// Mitsubishi GX Works2 project: TSUNE-14.10.2020_Q03UDV-FR   PLC: Q03UDV

PROGRAM MAIN
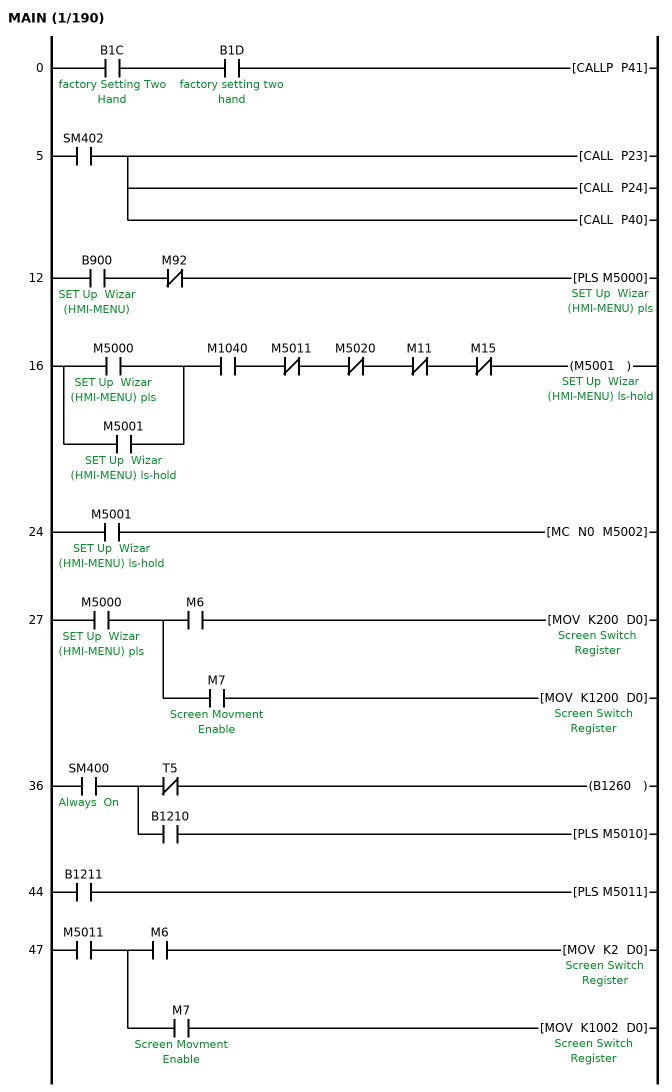
0     LD      B1C  ; factory Setting Two Hand
      AND     B1D  ; factory setting two hand
      CALLP   P41
5     LD      SM402
      CALL    P23
      CALL    P24
      CALL    P40
12    LD      B900  ; SET Up  Wizar  (HMI-MENU)
      ANI     M92
      PLS     M5000  ; SET Up  Wizar  (HMI-MENU) pls
16    LD      M5000  ; SET Up  Wizar  (HMI-MENU) pls
      OR      M5001  ; SET Up  Wizar (HMI-MENU) ls-hold
      AND     M1040
      ANI     M5011
      ANI     M5020
      ANI     M11
      ANI     M15
      OUT     M5001  ; SET Up  Wizar (HMI-MENU) ls-hold
24    LD      M5001  ; SET Up  Wizar (HMI-MENU) ls-hold
      MC      N0 M5002
27    LD      M5000  ; SET Up  Wizar  (HMI-MENU) pls
      MPS
      AND     M6
      MOV     K200 D0  ; Screen Switch Register
      MPP
      AND     M7  ; Screen Movment Enable
      MOV     K1200 D0
36    LD      SM400  ; Always  On
      MPS
      ANI     T5
      OUT     B1260
      MPP
      AND     B1210
      PLS     M5010
44    LD      B1211
      PLS     M5011
47    LD      M5011
      MPS
      AND     M6
      MOV     K2 D0
      MPP
      AND     M7  ; Screen Movment Enable
      MOV     K1002 D0
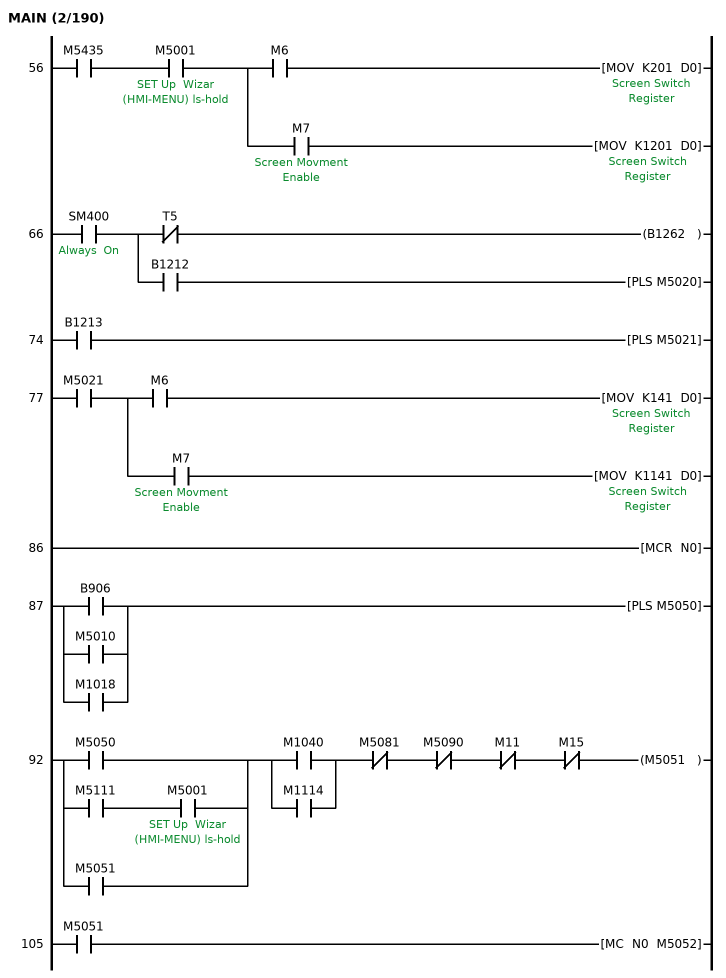
56    LD      M5435
      AND     M5001  ; SET Up  Wizar (HMI-MENU) ls-hold
      MPS
      AND     M6
      MOV     K201 D0
      MPP
      AND     M7  ; Screen Movment Enable
      MOV     K1201 D0
66    LD      SM400  ; Always  On
      MPS
      ANI     T5
      OUT     B1262
      MPP
      AND     B1212
      PLS     M5020
74    LD      B1213
      PLS     M5021
77    LD      M5021
      MPS
      AND     M6
      MOV     K141 D0
      MPP
      AND     M7  ; Screen Movment Enable
      MOV     K1141 D0
86    MCR     N0
87    LD      B906
      OR      M5010
      OR      M1018
      PLS     M5050
92    LD      M5050
      LD      M5111
      AND     M5001  ; SET Up  Wizar (HMI-MENU) ls-hold
      ORB
      OR      M5051
      LD      M1040
      OR      M1114
      ANB
      ANI     M5081
      ANI     M5090
      ANI     M11
      ANI     M15
      OUT     M5051
105   LD      M5051
      MC      N0 M5052
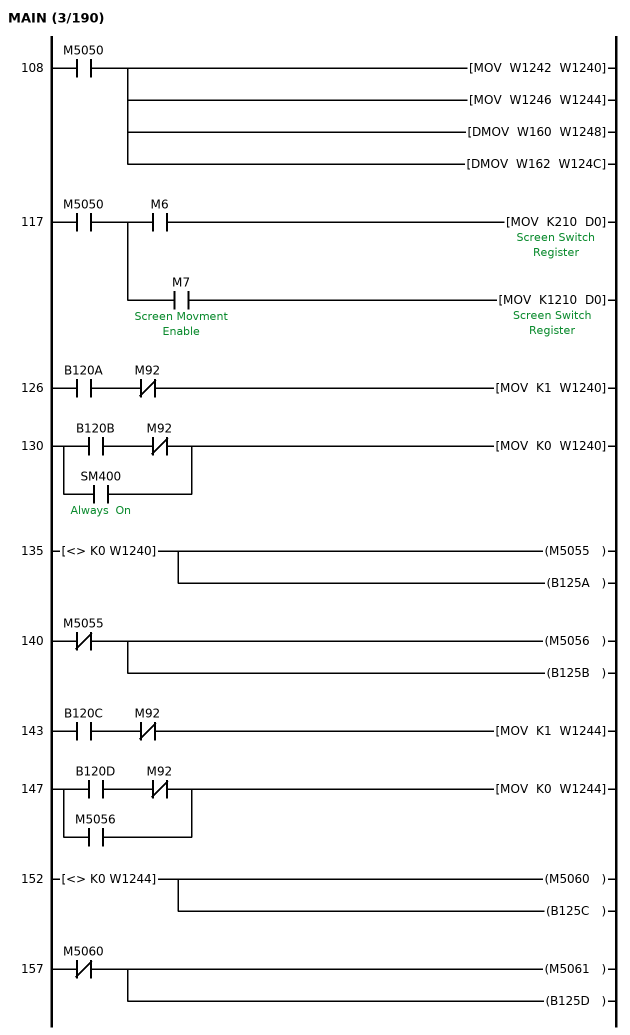
108   LD      M5050
      MOV     W1242 W1240
      MOV     W1246 W1244
      DMOV    W160 W1248
      DMOV    W162 W124C
117   LD      M5050
      MPS
      AND     M6
      MOV     K210 D0
      MPP
      AND     M7  ; Screen Movment Enable
      MOV     K1210 D0
126   LD      B120A
      ANI     M92
      MOV     K1 W1240
130   LD      B120B
      ANI     M92
      OR      SM400  ; Always  On
      MOV     K0 W1240
135   LD<>    K0 W1240
      OUT     M5055
      OUT     B125A
140   LDI     M5055
      OUT     M5056
      OUT     B125B
143   LD      B120C
      ANI     M92
      MOV     K1 W1244
147   LD      B120D
      ANI     M92
      OR      M5056
      MOV     K0 W1244
152   LD<>    K0 W1244
      OUT     M5060
      OUT     B125C
157   LDI     M5060
      OUT     M5061
      OUT     B125D
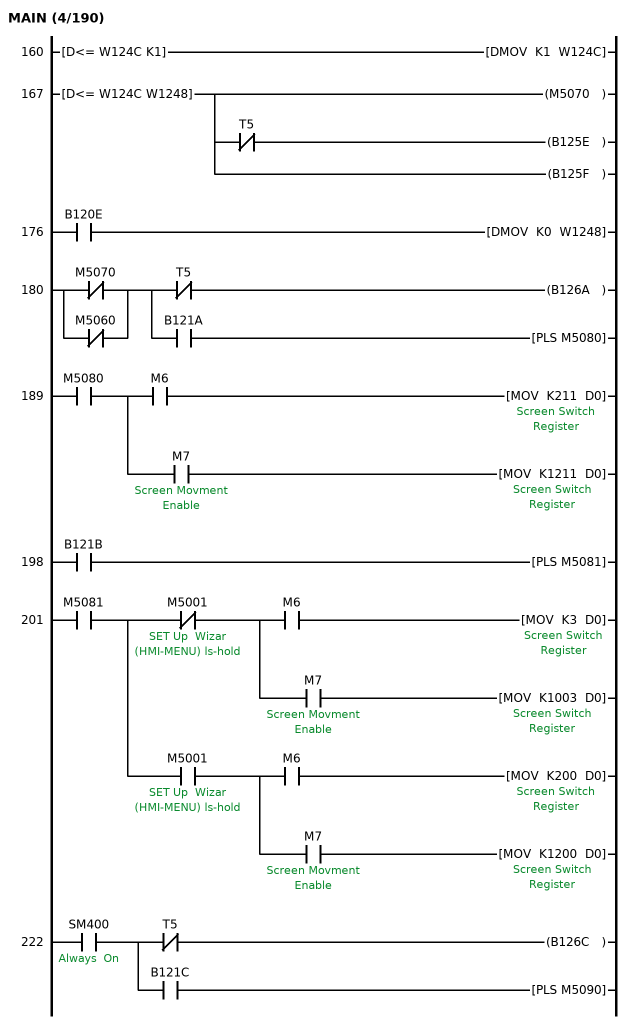
160   LDD<=   W124C K1
      DMOV    K1 W124C
167   LDD<=   W124C W1248
      OUT     M5070
      MPS
      ANI     T5
      OUT     B125E
      MPP
      OUT     B125F
176   LD      B120E
      DMOV    K0 W1248
180   LDI     M5070
      ORI     M5060
      MPS
      ANI     T5
      OUT     B126A
      MPP
      AND     B121A
      PLS     M5080
189   LD      M5080
      MPS
      AND     M6
      MOV     K211 D0
      MPP
      AND     M7  ; Screen Movment Enable
      MOV     K1211 D0
198   LD      B121B
      PLS     M5081
201   LD      M5081
      MPS
      ANI     M5001  ; SET Up  Wizar (HMI-MENU) ls-hold
      MPS
      AND     M6
      MOV     K3 D0
      MPP
      AND     M7  ; Screen Movment Enable
      MOV     K1003 D0
      MPP
      AND     M5001  ; SET Up  Wizar (HMI-MENU) ls-hold
      MPS
      AND     M6
      MOV     K200 D0
      MPP
      AND     M7  ; Screen Movment Enable
      MOV     K1200 D0
222   LD      SM400  ; Always  On
      MPS
      ANI     T5
      OUT     B126C
      MPP
      AND     B121C
      PLS     M5090
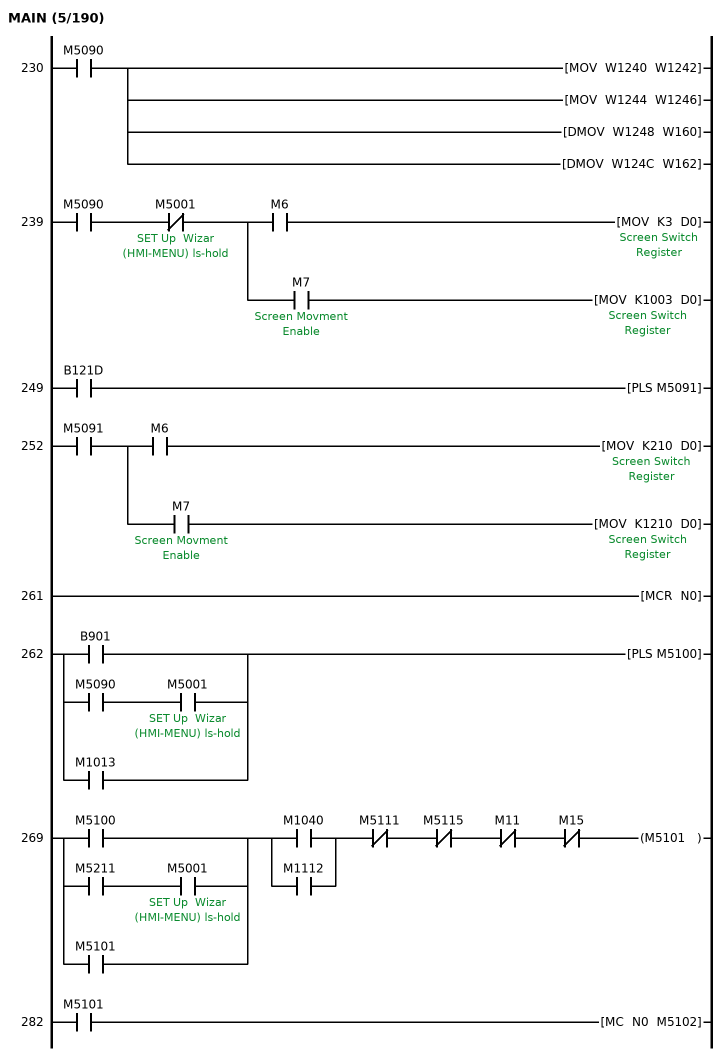
230   LD      M5090
      MOV     W1240 W1242
      MOV     W1244 W1246
      DMOV    W1248 W160
      DMOV    W124C W162
239   LD      M5090
      ANI     M5001  ; SET Up  Wizar (HMI-MENU) ls-hold
      MPS
      AND     M6
      MOV     K3 D0
      MPP
      AND     M7  ; Screen Movment Enable
      MOV     K1003 D0
249   LD      B121D
      PLS     M5091
252   LD      M5091
      MPS
      AND     M6
      MOV     K210 D0
      MPP
      AND     M7  ; Screen Movment Enable
      MOV     K1210 D0
261   MCR     N0
262   LD      B901
      LD      M5090
      AND     M5001  ; SET Up  Wizar (HMI-MENU) ls-hold
      ORB
      OR      M1013
      PLS     M5100
269   LD      M5100
      LD      M5211
      AND     M5001  ; SET Up  Wizar (HMI-MENU) ls-hold
      ORB
      OR      M5101
      LD      M1040
      OR      M1112
      ANB
      ANI     M5111
      ANI     M5115
      ANI     M11
      ANI     M15
      OUT     M5101
282   LD      M5101
      MC      N0 M5102
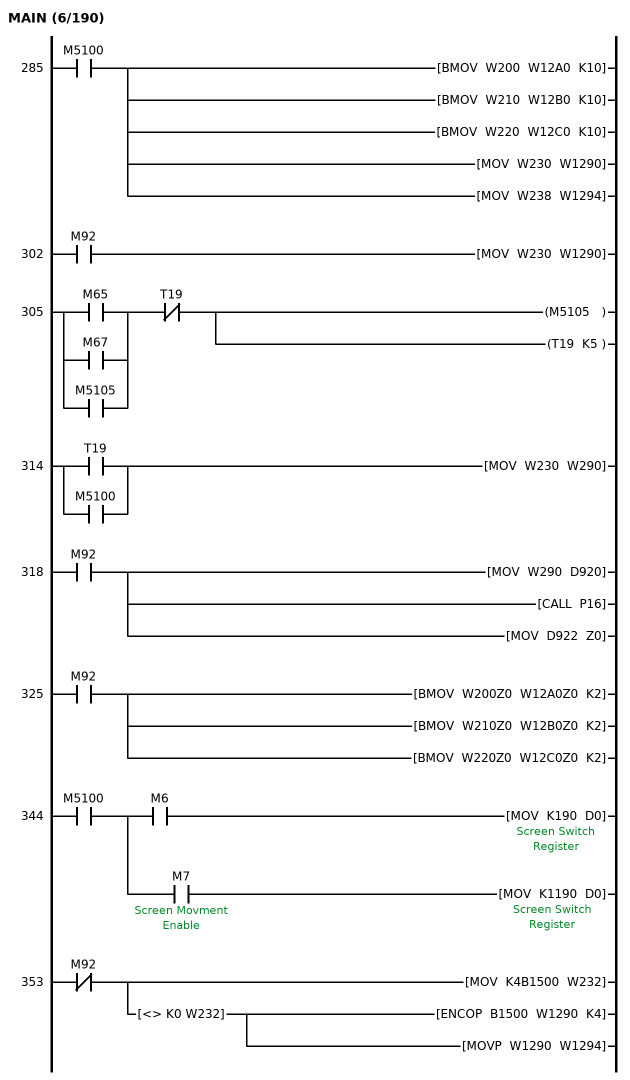
285   LD      M5100
      BMOV    W200 W12A0 K10
      BMOV    W210 W12B0 K10
      BMOV    W220 W12C0 K10
      MOV     W230 W1290
      MOV     W238 W1294
302   LD      M92
      MOV     W230 W1290
305   LD      M65
      OR      M67
      OR      M5105
      ANI     T19
      OUT     M5105
      OUT     T19 K5
314   LD      T19
      OR      M5100
      MOV     W230 W290
318   LD      M92
      MOV     W290 D920
      CALL    P16
      MOV     D922 Z0
325   LD      M92
      BMOV    W200Z0 W12A0Z0 K2
      BMOV    W210Z0 W12B0Z0 K2
      BMOV    W220Z0 W12C0Z0 K2
344   LD      M5100
      MPS
      AND     M6
      MOV     K190 D0
      MPP
      AND     M7  ; Screen Movment Enable
      MOV     K1190 D0
353   LDI     M92
      MOV     K4B1500 W232
      AND<>   K0 W232
      ENCOP   B1500 W1290 K4
      MOVP    W1290 W1294
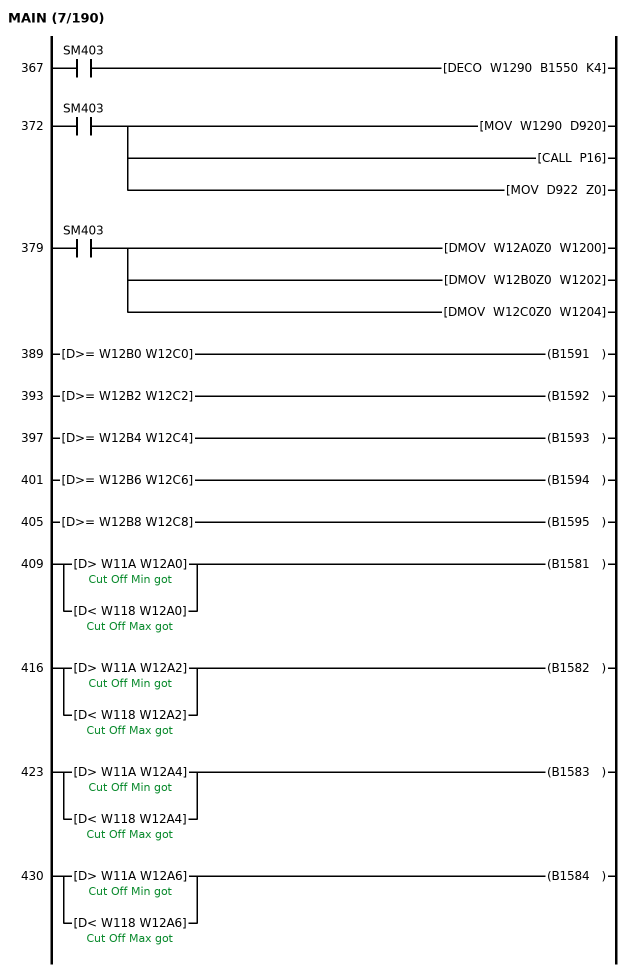
367   LD      SM403
      DECO    W1290 B1550 K4
372   LD      SM403
      MOV     W1290 D920
      CALL    P16
      MOV     D922 Z0
379   LD      SM403
      DMOV    W12A0Z0 W1200
      DMOV    W12B0Z0 W1202
      DMOV    W12C0Z0 W1204
389   LDD>=   W12B0 W12C0
      OUT     B1591
393   LDD>=   W12B2 W12C2
      OUT     B1592
397   LDD>=   W12B4 W12C4
      OUT     B1593
401   LDD>=   W12B6 W12C6
      OUT     B1594
405   LDD>=   W12B8 W12C8
      OUT     B1595
409   LDD>    W11A W12A0  ; Cut Off Min got
      ORD<    W118 W12A0  ; Cut Off Max got
      OUT     B1581
416   LDD>    W11A W12A2  ; Cut Off Min got
      ORD<    W118 W12A2  ; Cut Off Max got
      OUT     B1582
423   LDD>    W11A W12A4  ; Cut Off Min got
      ORD<    W118 W12A4  ; Cut Off Max got
      OUT     B1583
430   LDD>    W11A W12A6  ; Cut Off Min got
      ORD<    W118 W12A6  ; Cut Off Max got
      OUT     B1584
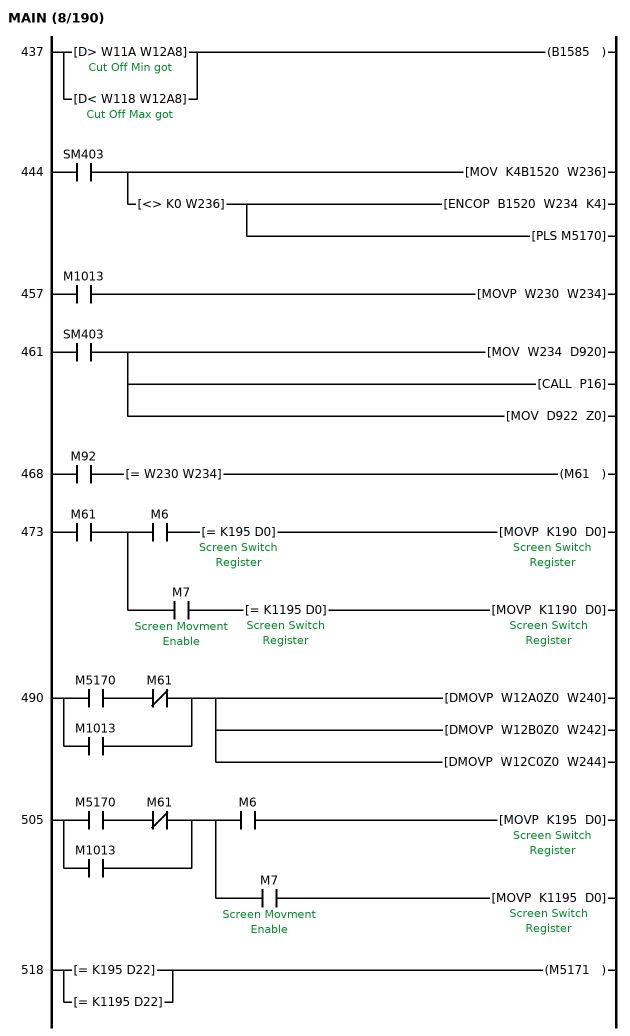
437   LDD>    W11A W12A8  ; Cut Off Min got
      ORD<    W118 W12A8  ; Cut Off Max got
      OUT     B1585
444   LD      SM403
      MOV     K4B1520 W236
      AND<>   K0 W236
      ENCOP   B1520 W234 K4
      PLS     M5170
457   LD      M1013
      MOVP    W230 W234
461   LD      SM403
      MOV     W234 D920
      CALL    P16
      MOV     D922 Z0
468   LD      M92
      AND=    W230 W234
      OUT     M61
473   LD      M61
      MPS
      AND     M6
      AND=    K195 D0  ; Screen Switch Register
      MOVP    K190 D0
      MPP
      AND     M7  ; Screen Movment Enable
      AND=    K1195 D0  ; Screen Switch Register
      MOVP    K1190 D0
490   LD      M5170
      ANI     M61
      OR      M1013
      DMOVP   W12A0Z0 W240
      DMOVP   W12B0Z0 W242
      DMOVP   W12C0Z0 W244
505   LD      M5170
      ANI     M61
      OR      M1013
      MPS
      AND     M6
      MOVP    K195 D0
      MPP
      AND     M7  ; Screen Movment Enable
      MOVP    K1195 D0
518   LD=     K195 D22
      OR=     K1195 D22
      OUT     M5171
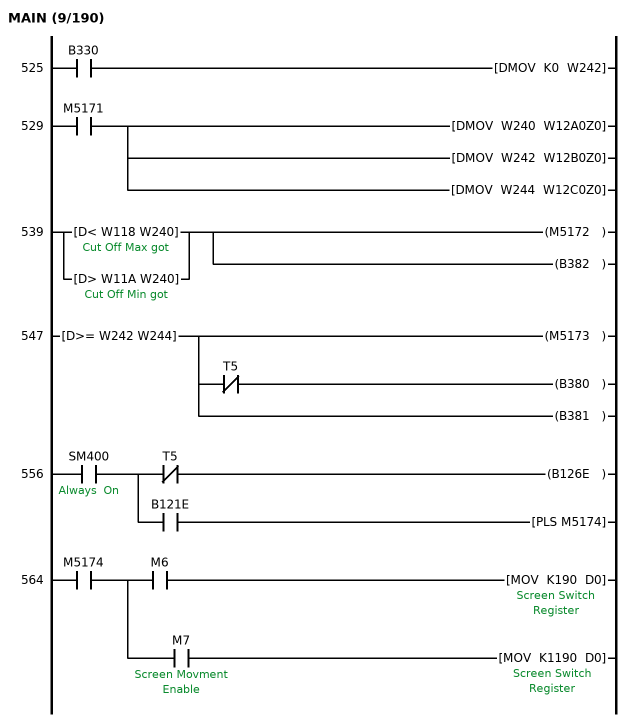
525   LD      B330
      DMOV    K0 W242
529   LD      M5171
      DMOV    W240 W12A0Z0
      DMOV    W242 W12B0Z0
      DMOV    W244 W12C0Z0
539   LDD<    W118 W240  ; Cut Off Max got
      ORD>    W11A W240  ; Cut Off Min got
      OUT     M5172
      OUT     B382
547   LDD>=   W242 W244
      OUT     M5173
      MPS
      ANI     T5
      OUT     B380
      MPP
      OUT     B381
556   LD      SM400  ; Always  On
      MPS
      ANI     T5
      OUT     B126E
      MPP
      AND     B121E
      PLS     M5174
564   LD      M5174
      MPS
      AND     M6
      MOV     K190 D0
      MPP
      AND     M7  ; Screen Movment Enable
      MOV     K1190 D0
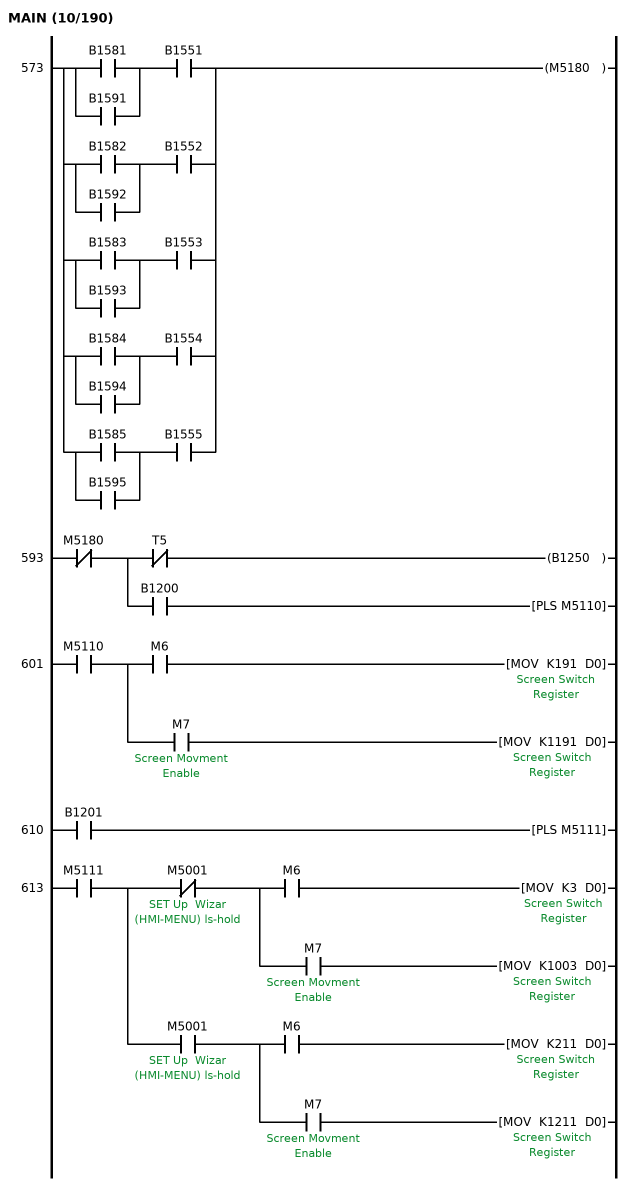
573   LD      B1581
      OR      B1591
      AND     B1551
      LD      B1582
      OR      B1592
      AND     B1552
      ORB
      LD      B1583
      OR      B1593
      AND     B1553
      ORB
      LD      B1584
      OR      B1594
      AND     B1554
      ORB
      LD      B1585
      OR      B1595
      AND     B1555
      ORB
      OUT     M5180
593   LDI     M5180
      MPS
      ANI     T5
      OUT     B1250
      MPP
      AND     B1200
      PLS     M5110
601   LD      M5110
      MPS
      AND     M6
      MOV     K191 D0
      MPP
      AND     M7  ; Screen Movment Enable
      MOV     K1191 D0
610   LD      B1201
      PLS     M5111
613   LD      M5111
      MPS
      ANI     M5001  ; SET Up  Wizar (HMI-MENU) ls-hold
      MPS
      AND     M6
      MOV     K3 D0
      MPP
      AND     M7  ; Screen Movment Enable
      MOV     K1003 D0
      MPP
      AND     M5001  ; SET Up  Wizar (HMI-MENU) ls-hold
      MPS
      AND     M6
      MOV     K211 D0
      MPP
      AND     M7  ; Screen Movment Enable
      MOV     K1211 D0
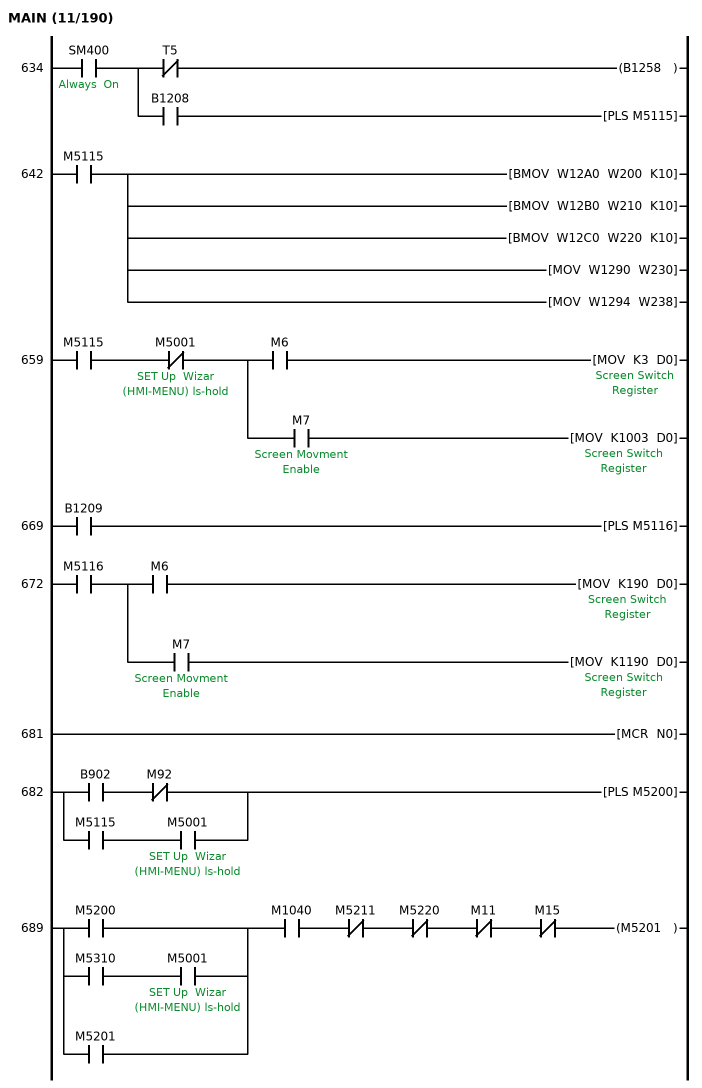
634   LD      SM400  ; Always  On
      MPS
      ANI     T5
      OUT     B1258
      MPP
      AND     B1208
      PLS     M5115
642   LD      M5115
      BMOV    W12A0 W200 K10
      BMOV    W12B0 W210 K10
      BMOV    W12C0 W220 K10
      MOV     W1290 W230
      MOV     W1294 W238
659   LD      M5115
      ANI     M5001  ; SET Up  Wizar (HMI-MENU) ls-hold
      MPS
      AND     M6
      MOV     K3 D0
      MPP
      AND     M7  ; Screen Movment Enable
      MOV     K1003 D0
669   LD      B1209
      PLS     M5116
672   LD      M5116
      MPS
      AND     M6
      MOV     K190 D0
      MPP
      AND     M7  ; Screen Movment Enable
      MOV     K1190 D0
681   MCR     N0
682   LD      B902
      ANI     M92
      LD      M5115
      AND     M5001  ; SET Up  Wizar (HMI-MENU) ls-hold
      ORB
      PLS     M5200
689   LD      M5200
      LD      M5310
      AND     M5001  ; SET Up  Wizar (HMI-MENU) ls-hold
      ORB
      OR      M5201
      AND     M1040
      ANI     M5211
      ANI     M5220
      ANI     M11
      ANI     M15
      OUT     M5201
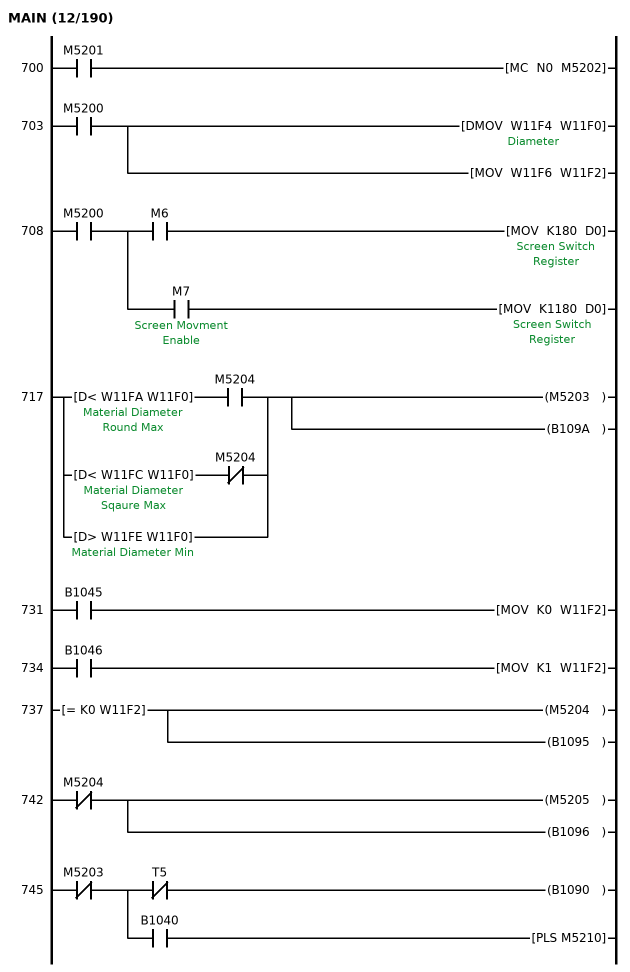
700   LD      M5201
      MC      N0 M5202
703   LD      M5200
      DMOV    W11F4 W11F0  ; Diameter
      MOV     W11F6 W11F2
708   LD      M5200
      MPS
      AND     M6
      MOV     K180 D0
      MPP
      AND     M7  ; Screen Movment Enable
      MOV     K1180 D0
717   LDD<    W11FA W11F0  ; Material Diameter Round Max
      AND     M5204
      LDD<    W11FC W11F0  ; Material Diameter Sqaure Max
      ANI     M5204
      ORB
      ORD>    W11FE W11F0  ; Material Diameter Min
      OUT     M5203
      OUT     B109A
731   LD      B1045
      MOV     K0 W11F2
734   LD      B1046
      MOV     K1 W11F2
737   LD=     K0 W11F2
      OUT     M5204
      OUT     B1095
742   LDI     M5204
      OUT     M5205
      OUT     B1096
745   LDI     M5203
      MPS
      ANI     T5
      OUT     B1090
      MPP
      AND     B1040
      PLS     M5210
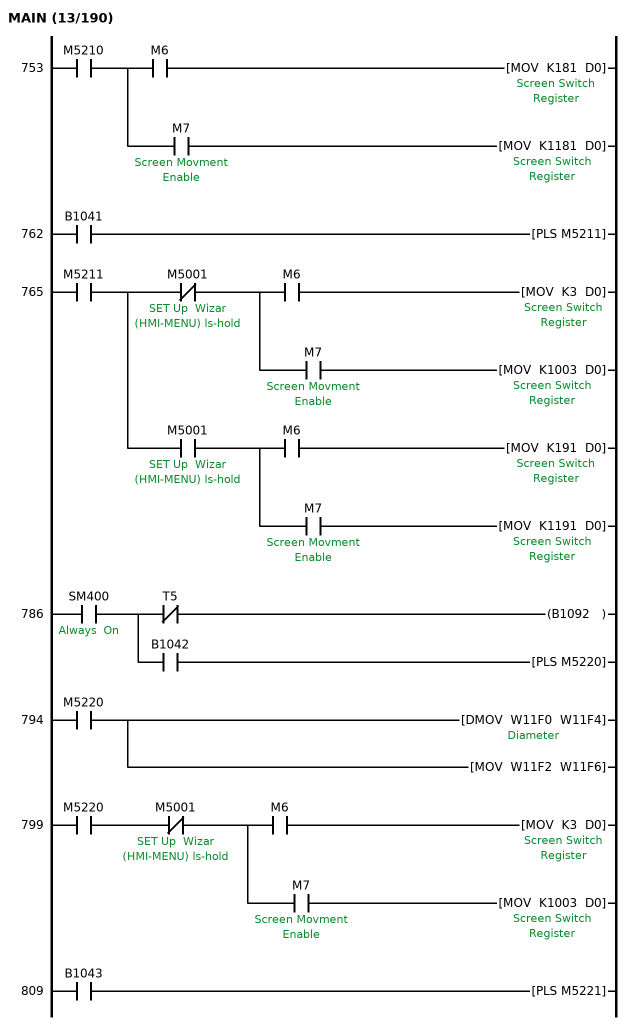
753   LD      M5210
      MPS
      AND     M6
      MOV     K181 D0
      MPP
      AND     M7  ; Screen Movment Enable
      MOV     K1181 D0
762   LD      B1041
      PLS     M5211
765   LD      M5211
      MPS
      ANI     M5001  ; SET Up  Wizar (HMI-MENU) ls-hold
      MPS
      AND     M6
      MOV     K3 D0
      MPP
      AND     M7  ; Screen Movment Enable
      MOV     K1003 D0
      MPP
      AND     M5001  ; SET Up  Wizar (HMI-MENU) ls-hold
      MPS
      AND     M6
      MOV     K191 D0
      MPP
      AND     M7  ; Screen Movment Enable
      MOV     K1191 D0
786   LD      SM400  ; Always  On
      MPS
      ANI     T5
      OUT     B1092
      MPP
      AND     B1042
      PLS     M5220
794   LD      M5220
      DMOV    W11F0 W11F4
      MOV     W11F2 W11F6
799   LD      M5220
      ANI     M5001  ; SET Up  Wizar (HMI-MENU) ls-hold
      MPS
      AND     M6
      MOV     K3 D0
      MPP
      AND     M7  ; Screen Movment Enable
      MOV     K1003 D0
809   LD      B1043
      PLS     M5221
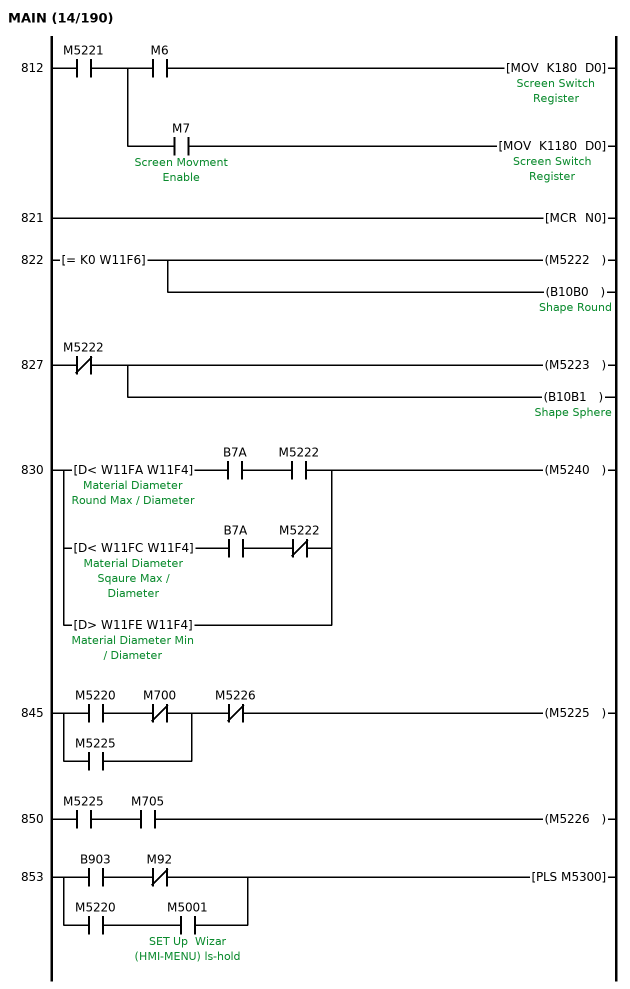
812   LD      M5221
      MPS
      AND     M6
      MOV     K180 D0
      MPP
      AND     M7  ; Screen Movment Enable
      MOV     K1180 D0
821   MCR     N0
822   LD=     K0 W11F6
      OUT     M5222
      OUT     B10B0  ; Shape Round
827   LDI     M5222
      OUT     M5223
      OUT     B10B1  ; Shape Sphere
830   LDD<    W11FA W11F4  ; Material Diameter Round Max / Diameter
      AND     B7A
      AND     M5222
      LDD<    W11FC W11F4  ; Material Diameter Sqaure Max / Diameter
      AND     B7A
      ANI     M5222
      ORB
      ORD>    W11FE W11F4  ; Material Diameter Min / Diameter
      OUT     M5240
845   LD      M5220
      ANI     M700
      OR      M5225
      ANI     M5226
      OUT     M5225
850   LD      M5225
      AND     M705
      OUT     M5226
853   LD      B903
      ANI     M92
      LD      M5220
      AND     M5001  ; SET Up  Wizar (HMI-MENU) ls-hold
      ORB
      PLS     M5300
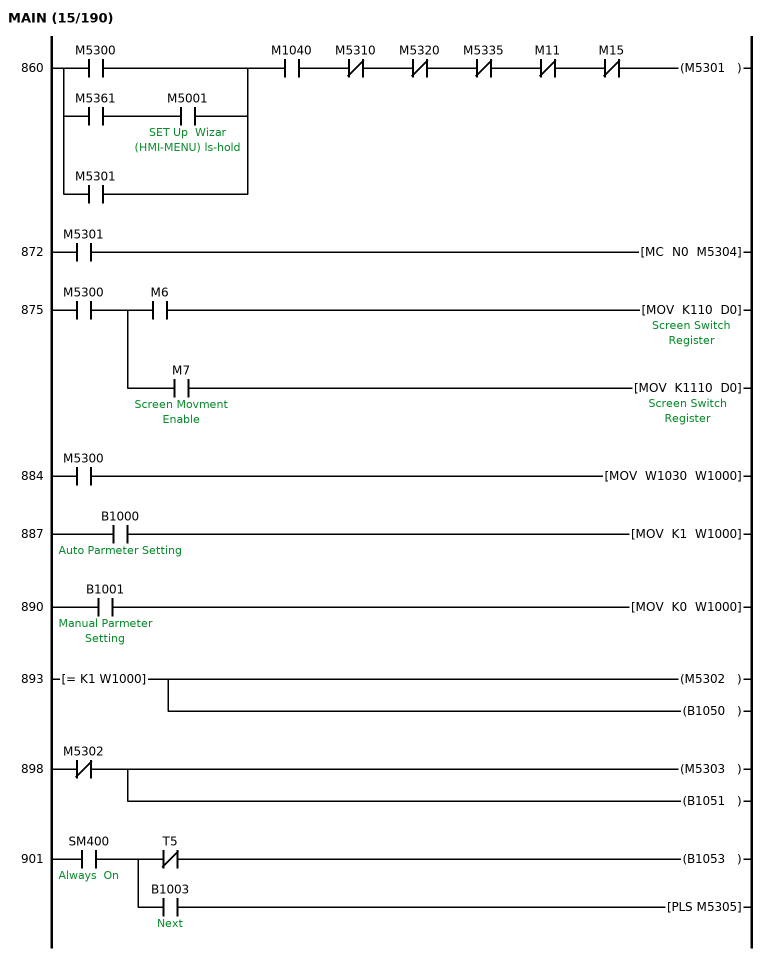
860   LD      M5300
      LD      M5361
      AND     M5001  ; SET Up  Wizar (HMI-MENU) ls-hold
      ORB
      OR      M5301
      AND     M1040
      ANI     M5310
      ANI     M5320
      ANI     M5335
      ANI     M11
      ANI     M15
      OUT     M5301
872   LD      M5301
      MC      N0 M5304
875   LD      M5300
      MPS
      AND     M6
      MOV     K110 D0
      MPP
      AND     M7  ; Screen Movment Enable
      MOV     K1110 D0
884   LD      M5300
      MOV     W1030 W1000
887   LD      B1000  ; Auto Parmeter Setting
      MOV     K1 W1000
890   LD      B1001  ; Manual Parmeter Setting
      MOV     K0 W1000
893   LD=     K1 W1000
      OUT     M5302
      OUT     B1050
898   LDI     M5302
      OUT     M5303
      OUT     B1051
901   LD      SM400  ; Always  On
      MPS
      ANI     T5
      OUT     B1053
      MPP
      AND     B1003  ; Next
      PLS     M5305
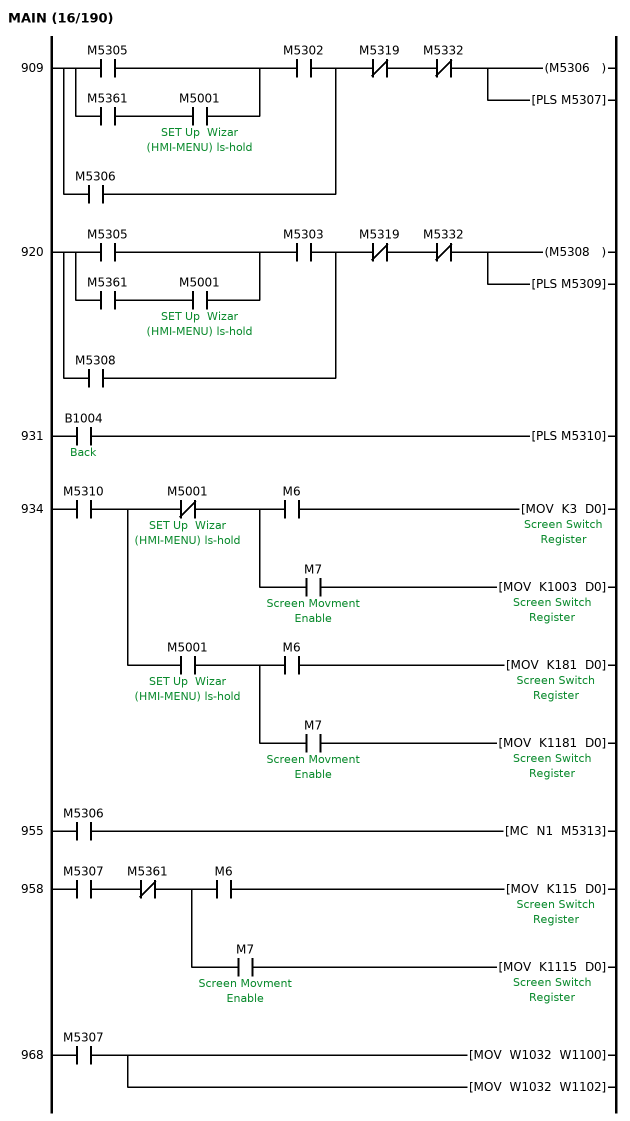
909   LD      M5305
      LD      M5361
      AND     M5001  ; SET Up  Wizar (HMI-MENU) ls-hold
      ORB
      AND     M5302
      OR      M5306
      ANI     M5319
      ANI     M5332
      OUT     M5306
      PLS     M5307
920   LD      M5305
      LD      M5361
      AND     M5001  ; SET Up  Wizar (HMI-MENU) ls-hold
      ORB
      AND     M5303
      OR      M5308
      ANI     M5319
      ANI     M5332
      OUT     M5308
      PLS     M5309
931   LD      B1004  ; Back
      PLS     M5310
934   LD      M5310
      MPS
      ANI     M5001  ; SET Up  Wizar (HMI-MENU) ls-hold
      MPS
      AND     M6
      MOV     K3 D0
      MPP
      AND     M7  ; Screen Movment Enable
      MOV     K1003 D0
      MPP
      AND     M5001  ; SET Up  Wizar (HMI-MENU) ls-hold
      MPS
      AND     M6
      MOV     K181 D0
      MPP
      AND     M7  ; Screen Movment Enable
      MOV     K1181 D0
955   LD      M5306
      MC      N1 M5313
958   LD      M5307
      ANI     M5361
      MPS
      AND     M6
      MOV     K115 D0
      MPP
      AND     M7  ; Screen Movment Enable
      MOV     K1115 D0
968   LD      M5307
      MOV     W1032 W1100
      MOV     W1032 W1102
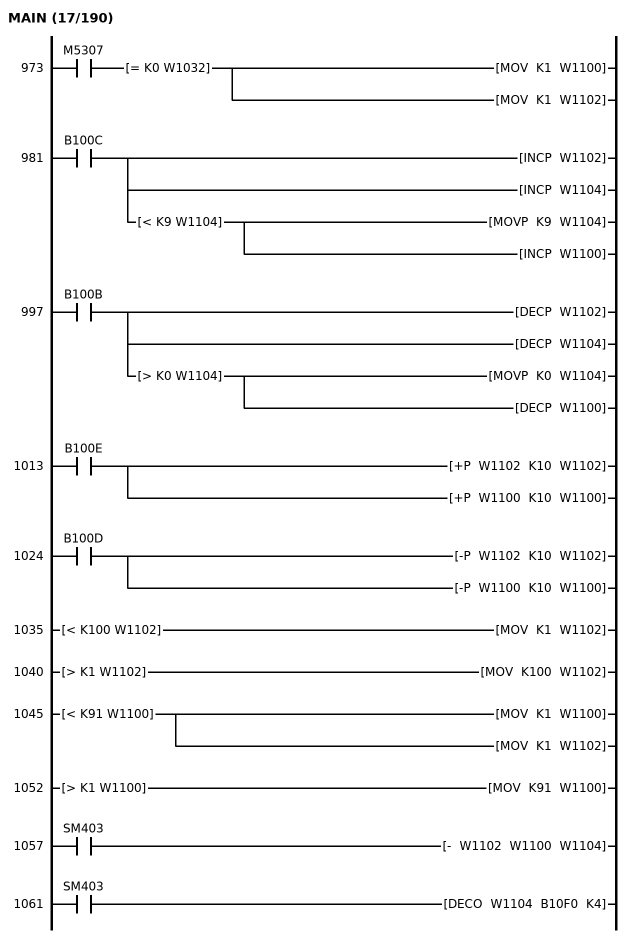
973   LD      M5307
      AND=    K0 W1032
      MOV     K1 W1100
      MOV     K1 W1102
981   LD      B100C
      INCP    W1102
      INCP    W1104
      AND<    K9 W1104
      MOVP    K9 W1104
      INCP    W1100
997   LD      B100B
      DECP    W1102
      DECP    W1104
      AND>    K0 W1104
      MOVP    K0 W1104
      DECP    W1100
1013  LD      B100E
      +P      W1102 K10 W1102
      +P      W1100 K10 W1100
1024  LD      B100D
      -P      W1102 K10 W1102
      -P      W1100 K10 W1100
1035  LD<     K100 W1102
      MOV     K1 W1102
1040  LD>     K1 W1102
      MOV     K100 W1102
1045  LD<     K91 W1100
      MOV     K1 W1100
      MOV     K1 W1102
1052  LD>     K1 W1100
      MOV     K91 W1100
1057  LD      SM403
      -       W1102 W1100 W1104
1061  LD      SM403
      DECO    W1104 B10F0 K4
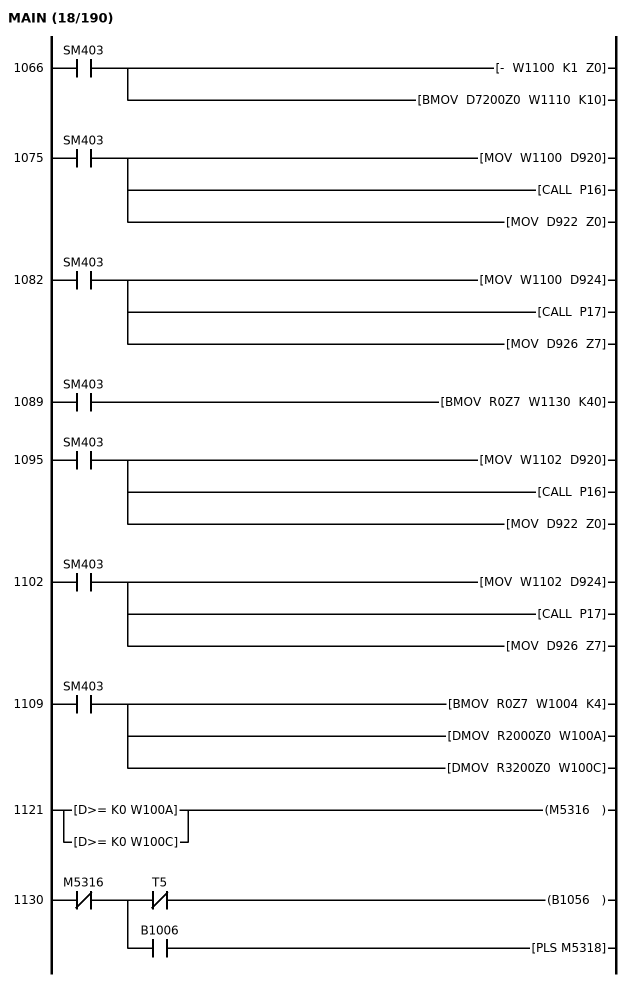
1066  LD      SM403
      -       W1100 K1 Z0
      BMOV    D7200Z0 W1110 K10
1075  LD      SM403
      MOV     W1100 D920
      CALL    P16
      MOV     D922 Z0
1082  LD      SM403
      MOV     W1100 D924
      CALL    P17
      MOV     D926 Z7
1089  LD      SM403
      BMOV    R0Z7 W1130 K40
1095  LD      SM403
      MOV     W1102 D920
      CALL    P16
      MOV     D922 Z0
1102  LD      SM403
      MOV     W1102 D924
      CALL    P17
      MOV     D926 Z7
1109  LD      SM403
      BMOV    R0Z7 W1004 K4
      DMOV    R2000Z0 W100A
      DMOV    R3200Z0 W100C
1121  LDD>=   K0 W100A
      ORD>=   K0 W100C
      OUT     M5316
1130  LDI     M5316
      MPS
      ANI     T5
      OUT     B1056
      MPP
      AND     B1006
      PLS     M5318
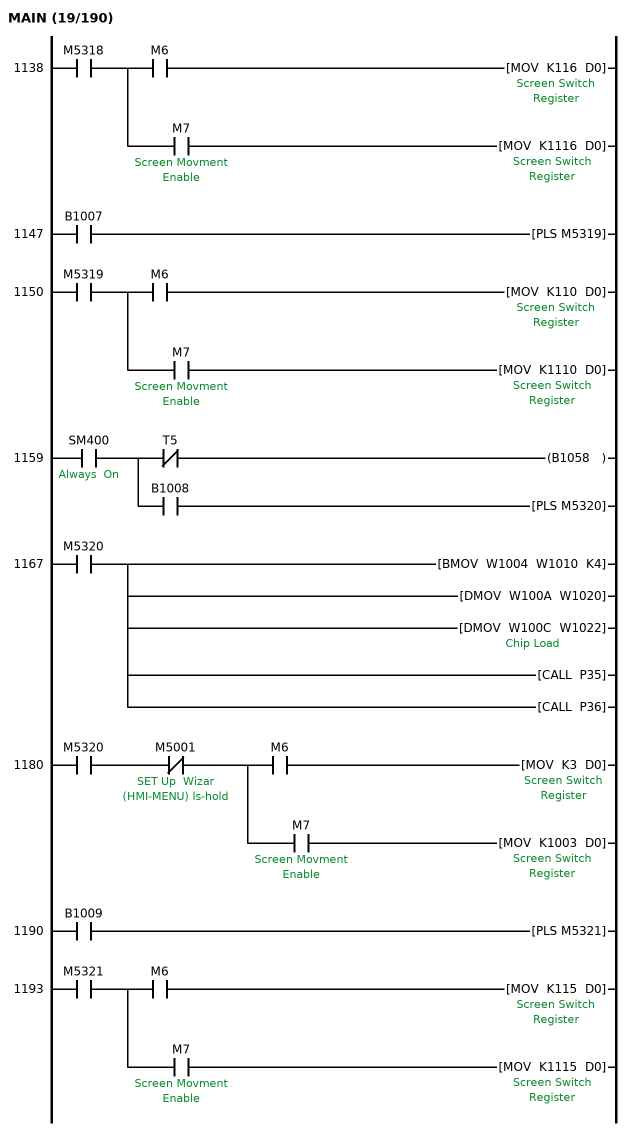
1138  LD      M5318
      MPS
      AND     M6
      MOV     K116 D0
      MPP
      AND     M7  ; Screen Movment Enable
      MOV     K1116 D0
1147  LD      B1007
      PLS     M5319
1150  LD      M5319
      MPS
      AND     M6
      MOV     K110 D0
      MPP
      AND     M7  ; Screen Movment Enable
      MOV     K1110 D0
1159  LD      SM400  ; Always  On
      MPS
      ANI     T5
      OUT     B1058
      MPP
      AND     B1008
      PLS     M5320
1167  LD      M5320
      BMOV    W1004 W1010 K4
      DMOV    W100A W1020
      DMOV    W100C W1022  ; Chip Load
      CALL    P35
      CALL    P36
1180  LD      M5320
      ANI     M5001  ; SET Up  Wizar (HMI-MENU) ls-hold
      MPS
      AND     M6
      MOV     K3 D0
      MPP
      AND     M7  ; Screen Movment Enable
      MOV     K1003 D0
1190  LD      B1009
      PLS     M5321
1193  LD      M5321
      MPS
      AND     M6
      MOV     K115 D0
      MPP
      AND     M7  ; Screen Movment Enable
      MOV     K1115 D0
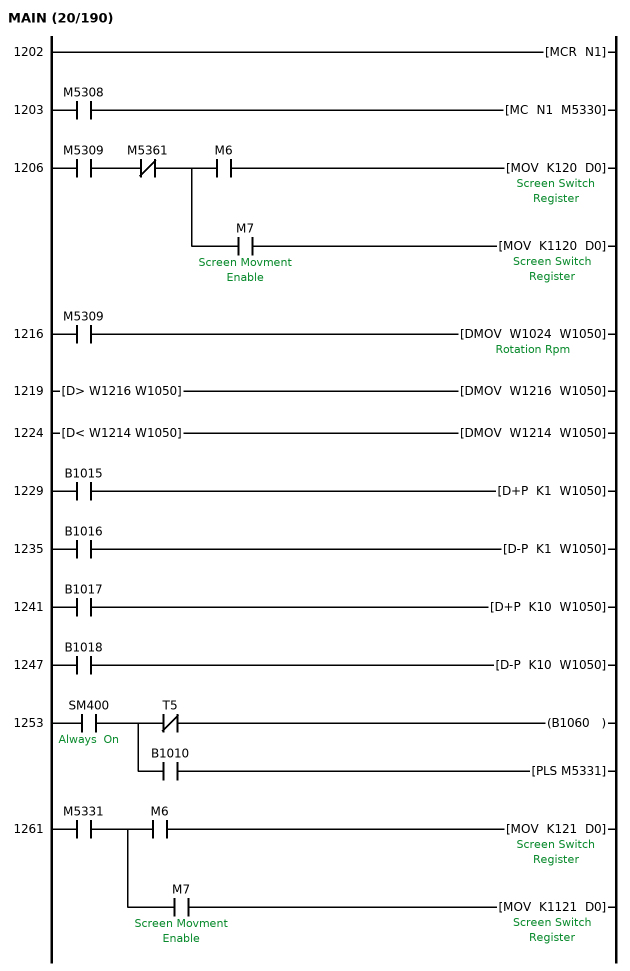
1202  MCR     N1
1203  LD      M5308
      MC      N1 M5330
1206  LD      M5309
      ANI     M5361
      MPS
      AND     M6
      MOV     K120 D0
      MPP
      AND     M7  ; Screen Movment Enable
      MOV     K1120 D0
1216  LD      M5309
      DMOV    W1024 W1050  ; Rotation Rpm
1219  LDD>    W1216 W1050
      DMOV    W1216 W1050
1224  LDD<    W1214 W1050
      DMOV    W1214 W1050
1229  LD      B1015
      D+P     K1 W1050
1235  LD      B1016
      D-P     K1 W1050
1241  LD      B1017
      D+P     K10 W1050
1247  LD      B1018
      D-P     K10 W1050
1253  LD      SM400  ; Always  On
      MPS
      ANI     T5
      OUT     B1060
      MPP
      AND     B1010
      PLS     M5331
1261  LD      M5331
      MPS
      AND     M6
      MOV     K121 D0
      MPP
      AND     M7  ; Screen Movment Enable
      MOV     K1121 D0
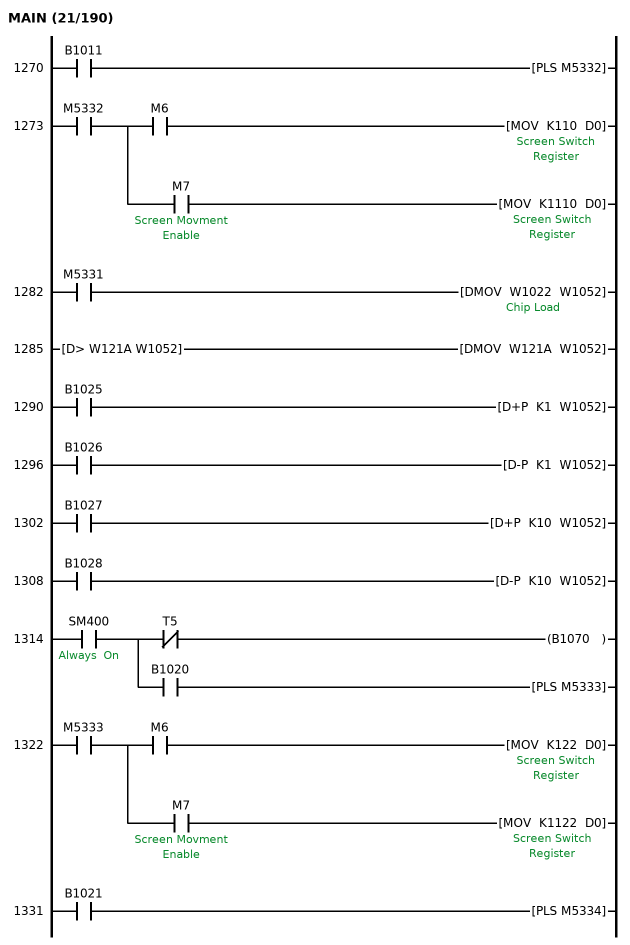
1270  LD      B1011
      PLS     M5332
1273  LD      M5332
      MPS
      AND     M6
      MOV     K110 D0
      MPP
      AND     M7  ; Screen Movment Enable
      MOV     K1110 D0
1282  LD      M5331
      DMOV    W1022 W1052
1285  LDD>    W121A W1052
      DMOV    W121A W1052
1290  LD      B1025
      D+P     K1 W1052
1296  LD      B1026
      D-P     K1 W1052
1302  LD      B1027
      D+P     K10 W1052
1308  LD      B1028
      D-P     K10 W1052
1314  LD      SM400  ; Always  On
      MPS
      ANI     T5
      OUT     B1070
      MPP
      AND     B1020
      PLS     M5333
1322  LD      M5333
      MPS
      AND     M6
      MOV     K122 D0
      MPP
      AND     M7  ; Screen Movment Enable
      MOV     K1122 D0
1331  LD      B1021
      PLS     M5334
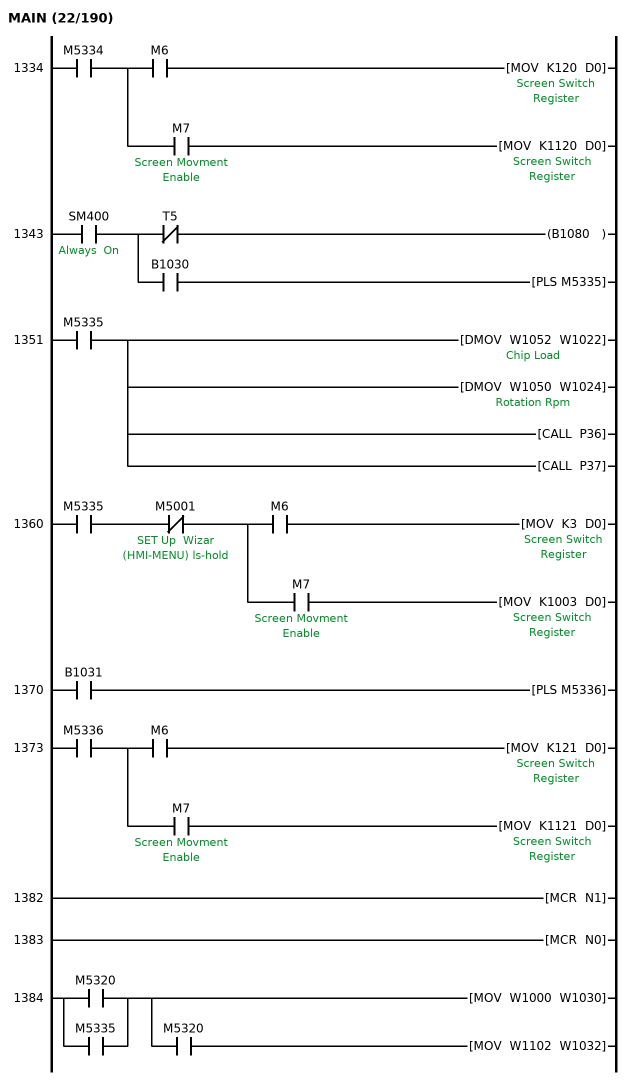
1334  LD      M5334
      MPS
      AND     M6
      MOV     K120 D0
      MPP
      AND     M7  ; Screen Movment Enable
      MOV     K1120 D0
1343  LD      SM400  ; Always  On
      MPS
      ANI     T5
      OUT     B1080
      MPP
      AND     B1030
      PLS     M5335
1351  LD      M5335
      DMOV    W1052 W1022
      DMOV    W1050 W1024
      CALL    P36
      CALL    P37
1360  LD      M5335
      ANI     M5001  ; SET Up  Wizar (HMI-MENU) ls-hold
      MPS
      AND     M6
      MOV     K3 D0
      MPP
      AND     M7  ; Screen Movment Enable
      MOV     K1003 D0
1370  LD      B1031
      PLS     M5336
1373  LD      M5336
      MPS
      AND     M6
      MOV     K121 D0
      MPP
      AND     M7  ; Screen Movment Enable
      MOV     K1121 D0
1382  MCR     N1
1383  MCR     N0
1384  LD      M5320
      OR      M5335
      MOV     W1000 W1030
      AND     M5320
      MOV     W1102 W1032
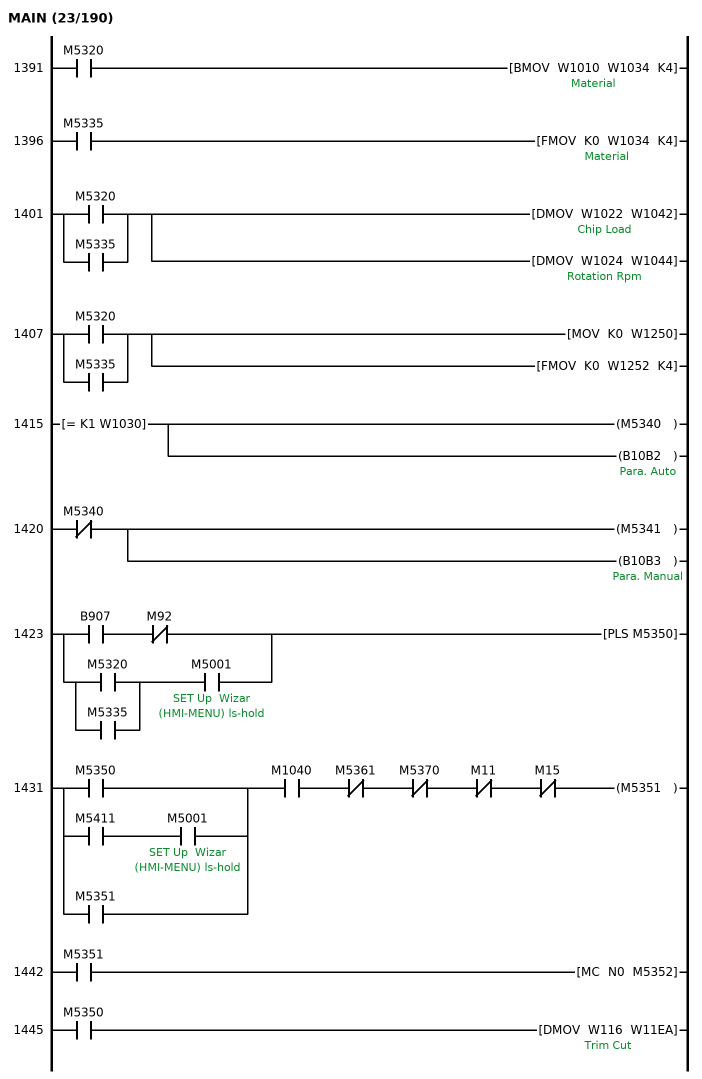
1391  LD      M5320
      BMOV    W1010 W1034 K4  ; Material
1396  LD      M5335
      FMOV    K0 W1034 K4
1401  LD      M5320
      OR      M5335
      DMOV    W1022 W1042
      DMOV    W1024 W1044
1407  LD      M5320
      OR      M5335
      MOV     K0 W1250
      FMOV    K0 W1252 K4
1415  LD=     K1 W1030
      OUT     M5340
      OUT     B10B2  ; Para. Auto
1420  LDI     M5340
      OUT     M5341
      OUT     B10B3  ; Para. Manual
1423  LD      B907
      ANI     M92
      LD      M5320
      OR      M5335
      AND     M5001  ; SET Up  Wizar (HMI-MENU) ls-hold
      ORB
      PLS     M5350
1431  LD      M5350
      LD      M5411
      AND     M5001  ; SET Up  Wizar (HMI-MENU) ls-hold
      ORB
      OR      M5351
      AND     M1040
      ANI     M5361
      ANI     M5370
      ANI     M11
      ANI     M15
      OUT     M5351
1442  LD      M5351
      MC      N0 M5352
1445  LD      M5350
      DMOV    W116 W11EA  ; Trim Cut
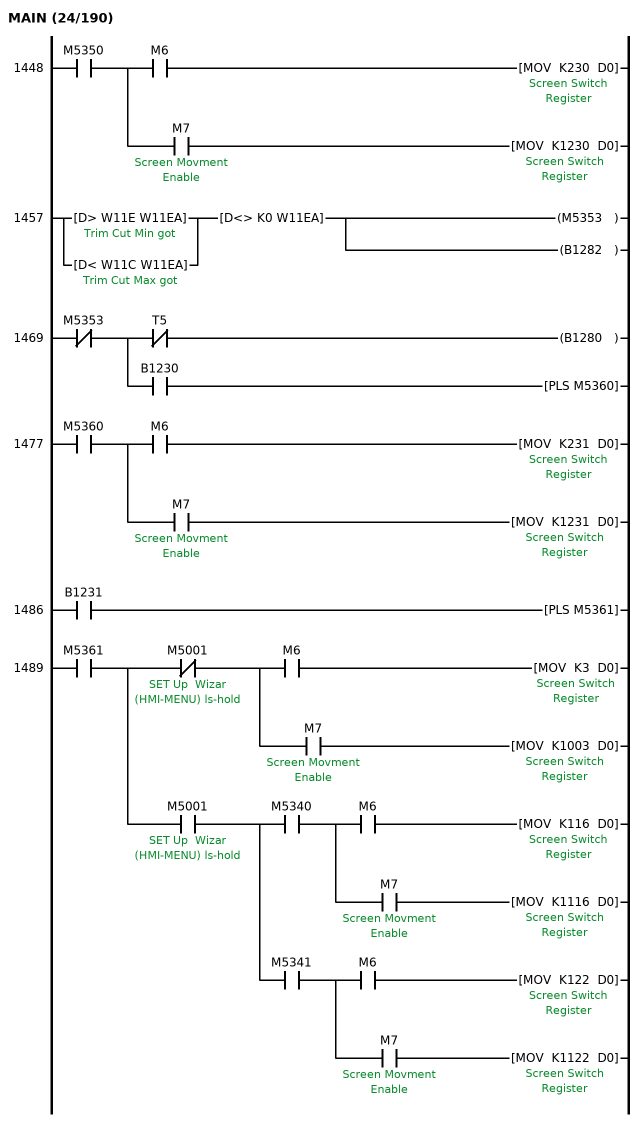
1448  LD      M5350
      MPS
      AND     M6
      MOV     K230 D0
      MPP
      AND     M7  ; Screen Movment Enable
      MOV     K1230 D0
1457  LDD>    W11E W11EA  ; Trim Cut Min got
      ORD<    W11C W11EA  ; Trim Cut Max got
      ANDD<>  K0 W11EA
      OUT     M5353
      OUT     B1282
1469  LDI     M5353
      MPS
      ANI     T5
      OUT     B1280
      MPP
      AND     B1230
      PLS     M5360
1477  LD      M5360
      MPS
      AND     M6
      MOV     K231 D0
      MPP
      AND     M7  ; Screen Movment Enable
      MOV     K1231 D0
1486  LD      B1231
      PLS     M5361
1489  LD      M5361
      MPS
      ANI     M5001  ; SET Up  Wizar (HMI-MENU) ls-hold
      MPS
      AND     M6
      MOV     K3 D0
      MPP
      AND     M7  ; Screen Movment Enable
      MOV     K1003 D0
      MPP
      AND     M5001  ; SET Up  Wizar (HMI-MENU) ls-hold
      MPS
      AND     M5340
      MPS
      AND     M6
      MOV     K116 D0
      MPP
      AND     M7  ; Screen Movment Enable
      MOV     K1116 D0
      MPP
      AND     M5341
      MPS
      AND     M6
      MOV     K122 D0
      MPP
      AND     M7  ; Screen Movment Enable
      MOV     K1122 D0
